{attribute 'qualified_only'}
TYPE E_ORDERTYPE :
(
    ASC := 0,
    DESC := 1
);
END_TYPE

(* stored: Version 1.1.0.1, ProductVersion 3.1.4024.9
   DUT E_ORDERTYPE: Id {a152bf14-65b8-4772-bc89-197714dcbf23} *)
